Staubli VAL3: language.pjx

Parameters version=s7.8.3 stackSize=5000 millimeterUnit=true
Program file=getLanguage.pgx
Program file=getYesNo.pgx
Program file=message.pgx
Program file=page.pgx
Program file=setLanguage.pgx
Data file=language.dtx
Library alias=language path=./chinese/chinese.pjx
